FUNCTION_BLOCK StampingProcess
VAR_INPUT
	MethodCall : BOOL;
	InputSensor: BOOL;
	StampingTime : TIME;
	NotAusSignal : BOOL;
	AutomaticMode: BOOL;
END_VAR
VAR_OUTPUT
	StampingProcess : BOOL;
END_VAR
VAR
//FlipFlop
	RS_StampingProcess: RS;
//Zeitverzögerung
	TOF_StampingTime: TOF;
//Flanke	
	R_TRIG_MethodCall: R_TRIG;
END_VAR
VAR // added by the converter: edge detectors and wires of the graphical bodies
    _w1 : BOOL;
END_VAR

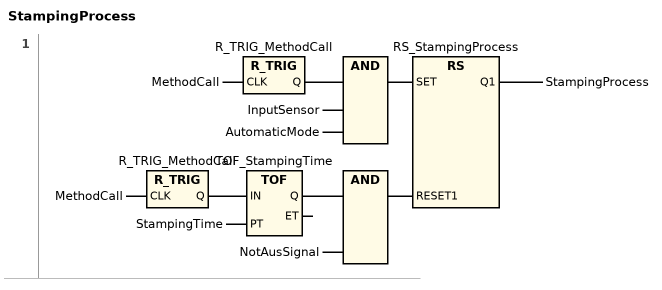
// NETWORK 1
R_TRIG_MethodCall(CLK := MethodCall); // R_TRIG
_w1 := R_TRIG_MethodCall.Q AND InputSensor AND AutomaticMode;
R_TRIG_MethodCall(CLK := MethodCall); // R_TRIG
TOF_StampingTime(IN := R_TRIG_MethodCall.Q, PT := StampingTime); // TOF
RS_StampingProcess(SET := _w1, RESET1 := TOF_StampingTime.Q AND NotAusSignal); // RS
StampingProcess := RS_StampingProcess.Q1;

END_FUNCTION_BLOCK

(* stored: Version 1.1.0.1, ProductVersion 3.1.4024.15
   POU StampingProcess: Id {fb2a4bc4-ff8d-4182-a54f-133db46eb046}, SpecialFunc None *)
